FUNCTION_BLOCK F_SEL_USINT (* selection (binary selection) *)
  (* Standard: 61131-3; Classification: standard selection function; Description: Copyright (c) 2012 TU Wien ACIN This program and the accompanying materials are made available under the terms of the Eclipse Public License 2.0 which is available at https://www.eclipse.org/legal/epl-2.0/ SPDX-License-Identifier: EPL-2.0 *)
  (* Version 1.0, 2012-03-25, Monika Wenger, TU Wien ACIN *)
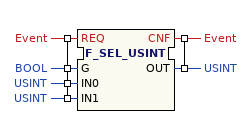
  EVENT_INPUT
    REQ WITH G, IN1, IN0; (* Service Request *)
  END_EVENT
  EVENT_OUTPUT
    CNF WITH OUT; (* Confirmation of Requested Service *)
  END_EVENT
  VAR_INPUT
    G : BOOL; (* Selelctor *)
    IN0 : USINT; (* Selectable input variable *)
    IN1 : USINT; (* Selectable input variable *)
  END_VAR
  VAR_OUTPUT
    OUT : USINT; (* Selected input *)
  END_VAR
END_FUNCTION_BLOCK
